{attribute 'GeneratedUsingTerminal: EK1100-0000-0018'}
{attribute addProperty BoxType "EK1100-0000-0018"}
{attribute addProperty Id "Beckhoff_EL3xxx_0030EK1122Beckhoff_EL3xxx_0030EK1122_BBE0797C2A_0001_EL3174_0030_0016EL3174_0E4717A052A_0002_EL3314_0030_0021EL3314_14E1817948A_0003_EL3681_0030_0021EL3681_B184412232A_0004_EL3201_0030_0022EL3201_F7A01EB921A_0005_EL3202_0030_0022EL3202_14BDD8A530A_0006_EL3356_0030_0025EL3356_BED8D8B728A_0007_EL3692_0030_0021EL3692_CD4ED2F352"}
{attribute addProperty CRC "518553542"}
{attribute addProperty Size "265"}
TYPE Beckhoff_EL3xxx_0030_1EE87FC6 EXTENDS EK1100_AB5A9467 :
STRUCT
	{attribute addProperty Name "Beckhoff_EL3xxx_0030EK1122"}
	Beckhoff_EL3xxx_0030EK1122 : Beckhoff_EL3xxx_0030EK1122_BBE0797C;
	{attribute addProperty Name "A_0001_EL3174_0030_0016"}
	A_0001_EL3174_0030_0016 : EL3174_0E4717A0;
	{attribute addProperty Name "A_0002_EL3314_0030_0021"}
	A_0002_EL3314_0030_0021 : EL3314_14E18179;
	{attribute addProperty Name "A_0003_EL3681_0030_0021"}
	A_0003_EL3681_0030_0021 : EL3681_B1844122;
	{attribute addProperty Name "A_0004_EL3201_0030_0022"}
	A_0004_EL3201_0030_0022 : EL3201_F7A01EB9;
	{attribute addProperty Name "A_0005_EL3202_0030_0022"}
	A_0005_EL3202_0030_0022 : EL3202_14BDD8A5;
	{attribute addProperty Name "A_0006_EL3356_0030_0025"}
	A_0006_EL3356_0030_0025 : EL3356_BED8D8B7;
	{attribute addProperty Name "A_0007_EL3692_0030_0021"}
	A_0007_EL3692_0030_0021 : EL3692_CD4ED2F3;
END_STRUCT
END_TYPE

(* stored: Version 1.2.0.0, ProductVersion 3.1.4024.9
   DUT Beckhoff_EL3xxx_0030_1EE87FC6: Id {df0815fa-0de7-4dec-b66c-29c83c726283} *)
